// TIA Portal V18 export
// export: Created 2023-08-11T09:04:57.8325312Z, ExportSetting WithDefaults, DisplayName Totally Integrated Automation Portal, DisplayVersion V18 Update 2, DisplayName TIA Portal Openness, DisplayVersion V18 Update 2, DisplayName TIA Portal Version Control Interface, DisplayVersion V18, DisplayName SINAMICS Startdrive Advanced, DisplayVersion V18, DisplayName SINAMICS Startdrive G130, G150, S120, S150, SINAMICS MV, S210, DisplayVersion V18, DisplayName SINAMICS Startdrive G110M, G120, G120C, G120D, G120P, G115D, DisplayVersion V18, DisplayName STEP 7 Professional, DisplayVersion V18 Update 2, DisplayName STEP 7 Safety, DisplayVersion V18, DisplayName WinCC Advanced / Unified PC, DisplayVersion V18 Update 2
FUNCTION_BLOCK "SinaSpeed2"   // FB1, SCL
{ S7_Optimized_Access := 'TRUE' }
VERSION : 0.1
// stored: AutoNumber true, IsIECCheckEnabled false, IsRetainMemResEnabled false, MemoryReserve 100, SetENOAutomatically false, UDAEnableTagReadback false
   VAR_INPUT
      EnableAxis : Bool;
      AckError : Bool;
      SpeedSp : Bool;
      RefSpeed : Bool;
      ConfigAxis : Bool;
      HWIDSTW : Bool;
      HWIDZSW : Bool;
      Input_1 : Int;
   END_VAR
   VAR_OUTPUT
      AxisEnabled : Bool;
      Lockout : Bool;
      ActVelocity : Bool;
      Error : Bool;
      Status : Bool;
      DiagId : Bool;
      InOut : Bool;
   END_VAR
   VAR
      STW1 : Bool;
      VelocitySP : Bool;
      ZSW1 : Bool;
      VelocityAV : Bool;
      testarvo : Bool;
   END_VAR
BEGIN
   #testarvo := 1;
END_FUNCTION_BLOCK
